{attribute addProperty BoxType "EL1258-0000-0017"}
{attribute addProperty Id "MTI_Inputs_10x_ChannelAT %I*ARRAY[0..7] OF MTI_Inputs_10x_Channel_7752F30830723840MTI_Outputs_ChannelAT %Q*ARRAY[0..7] OF MTI_Outputs_Channel_0FF822EF256320WcStateAT %I*WcState_F855686C1620InfoDataAT %I*InfoData_0BDED7BF144180"}
{attribute addProperty CRC "1659024344"}
{attribute addProperty SizeInBites "3488"}
{attribute addProperty SizeInBytes "436"}
TYPE EL1258_D5DBF8D7 :
STRUCT
	{attribute addProperty Name "MTI_Inputs_10x_Channel"}
	MTI_Inputs_10x_Channel : ARRAY[0..7] OF MTI_Inputs_10x_Channel_7752F308;
	{attribute addProperty Name "MTI_Outputs_Channel"}
	MTI_Outputs_Channel : ARRAY[0..7] OF MTI_Outputs_Channel_0FF822EF;
	{attribute addProperty Name "WcState"}
	WcState : WcState_F855686C;
	{attribute addProperty Name "InfoData"}
	InfoData : InfoData_0BDED7BF;
END_STRUCT
END_TYPE

(* stored: Version 1.2.0.0, ProductVersion 3.1.4024.9
   DUT EL1258_D5DBF8D7: Id {846ac0c8-537f-4064-9ce7-01f8360374ae} *)
